FUNCTION F_DebugUseEmuVizu : BOOL
VAR_IN_OUT
	SGref			: FB_ProBOXSG; //Reference to Switching group
	SG_Emuref		: FB_ProBOXSG_Emulation; //Reference to emulation switching group
END_VAR

//usage
// F_DebugUseEmuVizu(Groups.fbSG_001,GroupsEmulation.fbSG_001_Emulation)


SGref.HW_Inputs.AK.OpResetError		:= SGref.HW_Inputs.AK.OpResetError 	OR SG_Emuref.DebugResetButton;
SGref.HW_Inputs.AK.OpAutoOn			:= SGref.HW_Inputs.AK.OpAutoOn 		OR SG_Emuref.DebugStartButton;
SGref.HW_Inputs.AK.OpMcOn			:= SGref.HW_Inputs.AK.OpMcOn 		OR SG_Emuref.DebugMcOnButton;
SGref.HW_Inputs.AK.OpResetSafety	:= SGref.HW_Inputs.AK.OpResetSafety	OR SG_Emuref.DebugResetEmgButton;
SGref.HW_Inputs.AK.OpManAuto		:= SGref.HW_Inputs.AK.OpManAuto	AND NOT SG_Emuref.DebugManualModeSw;

END_FUNCTION

(* stored: Version 1.1.0.1, ProductVersion 3.1.4024.9
   POU F_DebugUseEmuVizu: Id {0a08792c-e8df-4790-87ef-4d0a9438c00d}, SpecialFunc None *)
